{attribute 'reflection'}
FUNCTION_BLOCK FB_ServiceBase EXTENDS FB_PackMLModeSet
VAR_INPUT
	Ctrl : REFERENCE TO ST_ServiceCtrl;
	Context : REFERENCE TO ST_ServiceContext;
	
	// The Module assigns a unique ID to this Service instance.
	ServiceId : T_ResourceOwnerId;
END_VAR

VAR_OUTPUT
	Status : ST_ServiceStatus;
END_VAR

VAR
	_CmdRequestOneShot : R_TRIG;
	_LastObservedPackMLState : E_PackMLState := E_PackMLState.Undefined;
	_ActiveExecuteSubStateRecord : UINT;
	
	{attribute 'instance-path'}
    {attribute 'noinit'}
	_Path : STRING;
END_VAR

METHOD PROTECTED H_GetExecuteSubState : UDINT
H_GetExecuteSubState := 0;
END_METHOD

METHOD PROTECTED H_GetExecuteSubStateName : STRING(80)
H_GetExecuteSubStateName := '';
END_METHOD

METHOD PROTECTED FINAL M_AddError : BOOL
VAR_INPUT
	MainErrorId : UDINT;
	SourceErrorId : UDINT;
	Message : STRING;
END_VAR

VAR
	nIndex : UINT;
	nFirstEmpty : UINT;
END_VAR
M_AddError := FALSE;
nFirstEmpty := 0;

FOR nIndex := 1 TO Param_Config.MaxServiceError DO
	IF Status.ErrorList[nIndex].MainErrorId = 0 THEN
		IF nFirstEmpty = 0 THEN
			nFirstEmpty := nIndex;
			EXIT;
		END_IF

	ELSIF Status.ErrorList[nIndex].MainErrorId = MainErrorId THEN
		// The same error event is already recorded for this task cycle.
		RETURN;
	END_IF
END_FOR

// Preserve the first ten errors; reject new errors when the list is full.
IF nFirstEmpty = 0 THEN
	RETURN;
END_IF

Status.ErrorList[nFirstEmpty].ModuleId := Context.ModuleId;
Status.ErrorList[nFirstEmpty].ServiceId := ServiceId;
Status.ErrorList[nFirstEmpty].MainErrorId := MainErrorId;
Status.ErrorList[nFirstEmpty].SourceErrorId := SourceErrorId;
Status.ErrorList[nFirstEmpty].Message := Message;
Status.ErrorList[nFirstEmpty].Path := _Path;
Status.ErrorList[nFirstEmpty].Severity := E_Severity.Alarm;
Status.ErrorList[nFirstEmpty].DateTime := Context.UtcDateTime;
Status.ErrorList[nFirstEmpty].Active := TRUE;
Status.ErrorList[nFirstEmpty].Acknowledged := FALSE;
Status.ErrorList[nFirstEmpty].OccurrenceCount := 1;
M_AddError := TRUE;
END_METHOD

METHOD PROTECTED FINAL M_ClearAllData
MEMSET(ADR(Status.Data), 0, SIZEOF(Status.Data));
END_METHOD

METHOD PROTECTED FINAL M_ClearAllError : BOOL
VAR_INPUT
END_VAR
MEMSET(ADR(Status.ErrorList), 0, SIZEOF(Status.ErrorList));
M_ClearAllError := TRUE;
END_METHOD

METHOD PROTECTED FINAL M_ClearData : BOOL
VAR_INPUT
	DataId : UDINT;
END_VAR
VAR
	nIndex : UINT;
END_VAR
M_ClearData := FALSE;
IF DataId = 0 THEN
	RETURN;
END_IF

FOR nIndex := 1 TO Param_Config.MaxServiceData DO
	IF Status.Data.DataList[nIndex].Id = DataId THEN
		MEMSET(ADR(Status.Data.DataList[nIndex]), 0, SIZEOF(Status.Data.DataList[nIndex]));
		IF Status.Data.Count > 0 THEN
			Status.Data.Count := Status.Data.Count - 1;
		END_IF
		Status.Data.Overflow := FALSE;
		M_ClearData := TRUE;
		RETURN;
	END_IF
END_FOR
END_METHOD

METHOD PRIVATE M_ClearExecuteSubStateStatus
MEMSET(ADR(Status.ExecuteSubState), 0, SIZEOF(Status.ExecuteSubState));
_ActiveExecuteSubStateRecord := 0;
END_METHOD

METHOD PRIVATE M_CloseExecuteSubStateRecord
IF (_ActiveExecuteSubStateRecord > 0)
	AND (_ActiveExecuteSubStateRecord <= Status.ExecuteSubState.RecordCount) THEN
	Status.ExecuteSubState.Records[_ActiveExecuteSubStateRecord].EndTimestamp := Context.UtcDateTime;
END_IF
_ActiveExecuteSubStateRecord := 0;
END_METHOD

METHOD PROTECTED FINAL M_UpdateData : BOOL
VAR_INPUT
	DataId : UDINT;
	Name : STRING(30);
	DataType : E_DescriptorType;
	Unit : STRING(10);
	Value : STRING(80);
END_VAR
VAR
	nIndex : UINT;
	nTargetIndex : UINT;
	nFirstEmpty : UINT;
END_VAR
M_UpdateData := FALSE;
IF DataId = 0 THEN
	RETURN;
END_IF

nTargetIndex := 0;
nFirstEmpty := 0;
FOR nIndex := 1 TO Param_Config.MaxServiceData DO
	IF Status.Data.DataList[nIndex].Id = DataId THEN
		nTargetIndex := nIndex;
		EXIT;
	ELSIF (Status.Data.DataList[nIndex].Id = 0) AND (nFirstEmpty = 0) THEN
		nFirstEmpty := nIndex;
	END_IF
END_FOR

IF nTargetIndex = 0 THEN
	IF nFirstEmpty = 0 THEN
		Status.Data.Overflow := TRUE;
		RETURN;
	END_IF
	nTargetIndex := nFirstEmpty;
	Status.Data.Count := Status.Data.Count + 1;
END_IF

Status.Data.DataList[nTargetIndex].Id := DataId;
Status.Data.DataList[nTargetIndex].Name := Name;
Status.Data.DataList[nTargetIndex].DataType := DataType;
Status.Data.DataList[nTargetIndex].Unit := Unit;
Status.Data.DataList[nTargetIndex].Value := Value;
M_UpdateData := TRUE;
END_METHOD

METHOD PRIVATE M_UpdateExecuteSubStateStatus
VAR_INPUT
	ExecuteActionEvaluated : BOOL;
END_VAR
VAR
	NewState : UDINT;
	NewRecordIndex : UINT;
END_VAR
IF PackMLOut.eStateCurrent <> E_PackMLState.Execute THEN
	M_CloseExecuteSubStateRecord();
	Status.ExecuteSubState.CurrentStep := 0;
	RETURN;
END_IF

// Entering Execute does not run H_OnExecute until the following Service scan.
// Do not sample a substate until an Execute action has actually been evaluated.
IF NOT ExecuteActionEvaluated THEN
	M_CloseExecuteSubStateRecord();
	Status.ExecuteSubState.CurrentStep := 0;
	RETURN;
END_IF

NewState := H_GetExecuteSubState();
IF NewState = Status.ExecuteSubState.CurrentStep THEN
	RETURN;
END_IF

M_CloseExecuteSubStateRecord();
Status.ExecuteSubState.CurrentStep := NewState;

// State zero means that the Service currently exposes no Execute substate.
IF NewState = 0 THEN
	RETURN;
END_IF

// Preserve the first records. CurrentState continues to update after overflow.
IF Status.ExecuteSubState.RecordCount >= Param_Config.MaxExecuteSubStateRecords THEN
	Status.ExecuteSubState.Overflow := TRUE;
	RETURN;
END_IF

NewRecordIndex := Status.ExecuteSubState.RecordCount + 1;
Status.ExecuteSubState.RecordCount := NewRecordIndex;
Status.ExecuteSubState.Records[NewRecordIndex].Step := NewState;
Status.ExecuteSubState.Records[NewRecordIndex].Name := H_GetExecuteSubStateName();
Status.ExecuteSubState.Records[NewRecordIndex].StartTimestamp := Context.UtcDateTime;
Status.ExecuteSubState.Records[NewRecordIndex].EndTimestamp := '';
_ActiveExecuteSubStateRecord := NewRecordIndex;
END_METHOD

METHOD PROTECTED FINAL M_UpdateService
VAR_INPUT
	CompletionBehavior : E_ServiceCompletionBehavior;
END_VAR
VAR
	bEnteredStarting : BOOL;
	PreviousPackMLState : E_PackMLState;
END_VAR
PreviousPackMLState := PackMLOut.eStateCurrent;
PackMLIn := Ctrl.PackMLIn;
SUPER^();

_CmdRequestOneShot(CLK:= PackMLIn.bCommandChangeRequest, Q=> );

// Starting may complete and enter Execute in the same scan. In that case,
// eStatePrevious still exposes the transient Starting state.
bEnteredStarting :=
	// Starting 執行超過1個 scan
	((PackMLOut.eStateCurrent = E_PackMLState.Starting)
		AND (_LastObservedPackMLState <> E_PackMLState.Starting))

	// Starting 在同一scan 就結束，即 _LastObservedPackMLState = Idle & PackMLOut.eStateCurrent = Execute
	OR ((PackMLOut.eStateCurrent = E_PackMLState.Execute)
		AND (PackMLOut.eStatePrevious = E_PackMLState.Starting)
		AND (_LastObservedPackMLState <> E_PackMLState.Starting)
		AND (_LastObservedPackMLState <> E_PackMLState.Execute));

IF bEnteredStarting THEN
	M_ClearExecuteSubStateStatus();
END_IF

// Update status.
Status.PackMLOut := PackMLOut;
M_UpdateExecuteSubStateStatus(
	ExecuteActionEvaluated := PreviousPackMLState = E_PackMLState.Execute);
Status.CompletionBehavior := CompletionBehavior;
Status.ServiceId := ServiceId;
IF _CmdRequestOneShot.Q THEN // Acknowledge to upper controller that command received
	Status.ResponseId := Ctrl.RequestId;
END_IF

_LastObservedPackMLState := PackMLOut.eStateCurrent;
END_METHOD

END_FUNCTION_BLOCK

(* stored: Version 1.1.0.1, ProductVersion 3.1.4026.18
   POU FB_ServiceBase: Id {db0b22da-7303-4462-851a-679b64cb7da9}, SpecialFunc None
   Folder Alarm: Id {739fe670-a0d7-4f1c-8e4d-40f9db23039d}
   Folder DataVariable: Id {3109a967-6bf3-43e8-a07e-99771f1a7861}
   Method H_GetExecuteSubState: Id {df111ed2-37f4-49f9-90f4-999a15583353}
   Method H_GetExecuteSubStateName: Id {9ebf9202-2dc7-4b2a-b268-d5c51d856bd3}
   Method M_AddError: Id {4e62615f-0e50-466e-9f56-aa0713d5e3ab}
   Method M_ClearAllData: Id {9ce708c8-fcc2-41b9-921d-4cf31cb789df}
   Method M_ClearAllError: Id {74a7f2fc-6f6d-42ad-ac47-9f603786b3c7}
   Method M_ClearData: Id {bda59455-e3cd-4825-a537-585be96d2e4e}
   Method M_ClearExecuteSubStateStatus: Id {c93def37-541e-45f2-9620-d2aa746a8f34}
   Method M_CloseExecuteSubStateRecord: Id {ae13a574-507c-49ec-b671-4310dd4e9261}
   Method M_UpdateData: Id {52f20474-69d8-45fd-9268-a22bd550dba9}
   Method M_UpdateExecuteSubStateStatus: Id {77545218-f183-4cc0-a793-b7c960834bdd}
   Method M_UpdateService: Id {8ae05b1d-81f7-4b0b-9f3f-42116c68a842} *)
